// TwinCAT 3 PLC project Test_PLC
// ProgramVersion: 3.1.4023.0
// libraries:
//   Tc2_Standard, * (Beckhoff Automation GmbH)
//   Tc2_System, * (Beckhoff Automation GmbH)
//   Tc3_Module, * (Beckhoff Automation GmbH)
// project tree:
//   DUTs/ DUT1.TcDUT, DUT2.TcDUT
//   / PlcTask.TcTTO
//   POUs/ Error.TcPOU, FB_Test.TcPOU, FB_Test2.TcPOU, MAIN.TcPOU
// real-time tasks:
//   TASK PlcTask: cycle T#10ms, priority 20, ADS port 350

CONFIGURATION Test_PLC
    RESOURCE PLC ON TwinCAT3
        TASK PlcTask(INTERVAL := T#10ms, PRIORITY := 20);
        PROGRAM MAIN WITH PlcTask : MAIN;
        PROGRAM Error WITH PlcTask : Error;
    END_RESOURCE
END_CONFIGURATION

// ---- DUTs/DUT1.TcDUT
TYPE DUT1 :
STRUCT
	i : INT;
	j : REAL;
	b : BOOL;
	
END_STRUCT
END_TYPE

// ---- DUTs/DUT2.TcDUT
TYPE DUT2 :
STRUCT
	i : INT;
	j : REAL;
	b : BOOL;
END_STRUCT
END_TYPE

// ---- POUs/MAIN.TcPOU
PROGRAM MAIN
VAR
	k :INT;
	
	s1 : DUT1;
	s2 : DUT2;
END_VAR

s1.b := TRUE;
s1.i := 99;
s1.j := 9.9;

s2 := s1;

END_PROGRAM

// ---- POUs/Error.TcPOU
PROGRAM Error
VAR_INPUT

END_VAR
VAR
		i : INT;
	fbTest : FB_Test;
END_VAR

i := fbTest.Prop;

END_PROGRAM

// ---- POUs/FB_Test.TcPOU
FUNCTION_BLOCK FB_Test
VAR_INPUT

END_VAR
VAR_OUTPUT
END_VAR
VAR
	j : INT;
	fbTest2 : FB_Test2;
END_VAR

PROPERTY PUBLIC Prop : INT
GET
Prop := j;
END_GET
END_PROPERTY

END_FUNCTION_BLOCK

// ---- POUs/FB_Test2.TcPOU
FUNCTION_BLOCK FB_Test2
VAR_INPUT
		i: INT;
END_VAR
VAR_OUTPUT
END_VAR
VAR

END_VAR

END_FUNCTION_BLOCK
